(* IEC 61131-3 sources: plc_simulator/services/codesys/POUs (part 2) *)

(* ---- FC_STC_ManualTask.st ---- *)
(* ===========================================================================================
 *  FC_STC_ManualTask — Execute manual transport tasks from gateway
 *
 *  Company : Galvatek part of the John Cockerill Group
 *  Author  : Jarmo Piipponen
 *  Created : 25.03.2026
 *
 * -------------------------------------------------------------------------------------------
 *  For each transporter, checks g_manual_task[vTi].Valid.
 *  If the transporter is idle (Phase=0), validates stations,
 *  calculates transfer time, and inserts a task into the queue
 *  (same pattern as FC_TSK_NoTreatment).
 *  Clears Valid after task is created, or on invalid input.
 *
 *  Called from FB_TSK_Scheduler vPhase 2200 (before NTT).
 *
 * ------------------------------------------------------------------------------------------
 *
 *  Changes:
 *
 *
 *
 *)

FUNCTION FC_STC_ManualTask : BOOL

(* Introduction of Variables ----------------------------------------------------------------*)

VAR_INPUT
  iTimeS                  : LINT;
END_VAR

VAR_IN_OUT
  ioTask                   : ARRAY[1..MAX_TRANSPORTERS] OF UDT_JC_TskQueueType;
END_VAR

VAR_EXTERNAL
  g_manual_task             : ARRAY[1..MAX_TRANSPORTERS] OF UDT_JC_ManualTaskType;
  g_transporter             : ARRAY[1..MAX_TRANSPORTERS] OF UDT_TransporterStatusType;
  g_move                    : ARRAY[1..MAX_TRANSPORTERS] OF UDT_JC_MoveTimesType;
  g_unit                    : ARRAY[1..MAX_UNITS] OF UDT_JC_UnitType;
  Stations                  : ARRAY[MIN_STATION_INDEX..MAX_STATION_INDEX] OF UDT_StationType;
  Transporters              : ARRAY[0..MAX_TRANSPORTERS] OF UDT_TransporterType;
END_VAR

VAR_EXTERNAL CONSTANT
  MAX_TASK_QUEUE            : INT;
  MAX_UNITS                 : INT;
  USED                      : INT;
END_VAR

VAR
  vTi                        : INT;
  vAi                        : INT;
  vSh                        : INT;
  vLift                      : INT;
  vSink                      : INT;
  vCovers                    : BOOL;
  vTransPos                 : INT;
  vTmpMove                  : UDT_JC_MoveTimesType;
  vXferS                    : REAL;
  vTravelToLiftS          : REAL;
  vTaskStart                : LINT;
  vTaskEnd                  : LINT;
END_VAR

FC_STC_ManualTask := TRUE;

FOR vTi := 1 TO MAX_TRANSPORTERS DO
  IF NOT g_manual_task[vTi].Valid THEN
    CONTINUE;
  END_IF;

  vLift := g_manual_task[vTi].LiftStation;
  vSink := g_manual_task[vTi].SinkStation;

  (* Validate station range *)
  IF vLift < MIN_STATION_INDEX OR vLift > MAX_STATION_INDEX
     OR vSink < MIN_STATION_INDEX OR vSink > MAX_STATION_INDEX
     OR vLift = vSink THEN
    g_manual_task[vTi].Valid := FALSE;
    CONTINUE;
  END_IF;

  (* Transporter must be active and idle *)
  (* Transporter must be active and idle or in move-away *)
  IF NOT g_transporter[vTi].IsActive THEN
    CONTINUE;
  END_IF;
  IF g_transporter[vTi].Phase <> 0
     AND NOT (g_transporter[vTi].Phase = 1 AND g_transporter[vTi].Status = 3) THEN
    CONTINUE;  (* keep Valid — retry next cycle *)
  END_IF;

  (* Check vLift station is within transporter TaskArea *)
  vCovers := FALSE;
  FOR vAi := 1 TO 4 DO
    IF Transporters[vTi].TaskArea[vAi].MinLift > 0
       OR Transporters[vTi].TaskArea[vAi].MaxLift > 0 THEN
      IF vLift >= Transporters[vTi].TaskArea[vAi].MinLift
         AND vLift <= Transporters[vTi].TaskArea[vAi].MaxLift THEN
        vCovers := TRUE;
      END_IF;
    END_IF;
  END_FOR;

  IF NOT vCovers THEN
    g_manual_task[vTi].Valid := FALSE;
    CONTINUE;
  END_IF;

  (* Calculate transfer time *)
  vTmpMove := g_move[vTi];
  vXferS := FC_STC_CalcTransferTime(
    iFromStn            := vLift,
    iToStn              := vSink,
    iMove                := vTmpMove,
    iFromDroppingX10   := Stations[vLift].DrippingTime,
    iToDeviceDelayX10 := Stations[vSink].DeviceDelay,
    iDripTrayDelayX10 := Transporters[vTi].DripTrayDelay);

  (* Calculate vTravel-to-vLift: time for transporter to reach vLift station *)
  vTravelToLiftS := 0.0;
  vTransPos := g_transporter[vTi].CurrentStation;
  IF vTransPos > 0 AND vTransPos <> vLift THEN
    vTravelToLiftS := FC_STC_CalcHorizontalTravel(
      iFromStn := vTransPos,
      iToStn   := vLift,
      iMove     := vTmpMove);
  END_IF;

  vTaskStart := iTimeS + REAL_TO_LINT(vTravelToLiftS);
  vTaskEnd   := vTaskStart + REAL_TO_LINT(vXferS);

  (* Check vSink station is free — no unit occupying it *)
  vCovers := TRUE;  (* reuse variable as vSinkFree flag *)
  FOR vSh := 1 TO MAX_UNITS DO
    IF g_unit[vSh].Location = vSink AND g_unit[vSh].Status = USED THEN
      vCovers := FALSE;
    END_IF;
  END_FOR;
  IF NOT vCovers THEN
    g_manual_task[vTi].Valid := FALSE;
    CONTINUE;
  END_IF;

  (* Insert task at queue position 1 *)
  IF ioTask[vTi].Count < MAX_TASK_QUEUE THEN
    FOR vSh := ioTask[vTi].Count TO 1 BY -1 DO
      ioTask[vTi].Queue[vSh + 1] := ioTask[vTi].Queue[vSh];
    END_FOR;
    ioTask[vTi].Queue[1].Unit              := 0;
    ioTask[vTi].Queue[1].Stage             := 0;
    ioTask[vTi].Queue[1].LiftStationTarget := vLift;
    ioTask[vTi].Queue[1].SinkStationTarget := vSink;
    ioTask[vTi].Queue[1].StartTime         := vTaskStart;
    ioTask[vTi].Queue[1].FinishTime        := vTaskEnd;
    ioTask[vTi].Queue[1].CalcTime          := 0;
    ioTask[vTi].Queue[1].MinTime           := 0;
    ioTask[vTi].Queue[1].MaxTime           := 0;
    ioTask[vTi].Queue[1].NttPrimary        := 0;
    ioTask[vTi].Count := ioTask[vTi].Count + 1;
  END_IF;

  g_manual_task[vTi].Valid := FALSE;
END_FOR;

END_FUNCTION

(* ---- FC_STC_NoTreatmentStates.st ---- *)
(* ===========================================================================================
 *  FC_STC_NoTreatmentStates — Non-treatment target state management
 *
 *  Company : Galvatek part of the John Cockerill Group
 *  Author  : Jarmo Piipponen
 *  Created : 25.03.2026
 *
 * -------------------------------------------------------------------------------------------
 *  Manages non-treatment target states for all units.
 *
 *  Structure:
 *  Pass 0 — SNAPSHOT: read unit/batch/station state into vSnap[]
 *  Section 1 — PROCESSED: mark last-stage units as PROCESSED
 *  Section 2 — TO_AVOID: clear occupied next-stage stations
 *  Section 3 — TO_LOADING: route one empty unit to loading
 *
 *  ------------------------------------------------------------------------------------------
 *
 *  Changes:
 *
 *
 *
 *)

FUNCTION FC_STC_NoTreatmentStates : BOOL

(* Introduction of Variables ----------------------------------------------------------------*)

VAR_EXTERNAL CONSTANT
    MAX_UNITS             : INT;
    MAX_STEPS_PER_PROGRAM : INT;
    MAX_STATIONS_PER_STEP : INT;
    MIN_STATION_INDEX     : INT;
    MAX_STATION_INDEX     : INT;
    IN_PROCESS            : INT;
    PROCESSED             : INT;
    NOT_USED              : INT;
    TO_NONE               : INT;
    TO_UNLOAD             : INT;
    TO_AVOID              : INT;
    TO_LOADING            : INT;
    USED                  : INT;
    OP_BUFFER             : INT;
    OP_BUFFER_PROCESSED   : INT;
    OP_LOADING            : INT;
    OP_LOADING_UNLOADING  : INT;
END_VAR

VAR_EXTERNAL
  gUnit              : ARRAY[1..MAX_UNITS] OF UDT_JC_UnitType;
  gBatch             : ARRAY[1..MAX_UNITS] OF UDT_BatchType;
  TreatmentPrograms  : ARRAY[1..MAX_UNITS] OF UDT_TreatmentProgramType;
  Stations           : ARRAY[MIN_STATION_INDEX..MAX_STATION_INDEX] OF UDT_StationType;
  gStationOccupancy  : ARRAY[1..MAX_STATION_INDEX] OF UDT_JC_UnitAtStationType;
  gTimeS             : LINT;
  gProductionQueue   : INT;
  gEventPending      : UDT_JC_EventMsgType;
  gEventPendingValid : BOOL;
END_VAR

VAR
  (* Snapshot *)
  vSnap       : ARRAY[1..MAX_UNITS] OF UDT_JC_UnitSnapType;
  vU          : INT;        (* unit loop index *)
  vHasLoading : BOOL;       (* any unit vAlready has TO_LOADING *)
  (* Section 1+2 *)
  vP          : INT;        (* parallel station loop *)
  vNextStn    : INT;        (* next stage station *)
  vOccUid     : INT;        (* unit_id at an occupied station *)
  vFreeFound  : BOOL;       (* any next-stage station is free *)
  vAvoidUid   : INT;        (* unit to mark TO_AVOID *)
  (* Section 3 *)
  vLoadFree   : BOOL;       (* a loading station is free *)
  vLoadUid    : INT;        (* best candidate for TO_LOADING *)
  vLoadInBuf  : BOOL;       (* current candidate is in buffer *)
  vStk        : INT;        (* station loop *)
  vOp         : INT;        (* station operation code *)
END_VAR

  (* ════════════════════════════════════════════════════════════
     Pass 0 — SNAPSHOT: collect per-unit state in one pass
     ════════════════════════════════════════════════════════════ *)
  vHasLoading := FALSE;

  FOR vU := 1 TO MAX_UNITS DO
    vSnap[vU].IsActive := gUnit[vU].Status <> NOT_USED;
    IF NOT vSnap[vU].IsActive THEN
      CONTINUE;
    END_IF;

    vSnap[vU].Location       := gUnit[vU].Location;
    vSnap[vU].Target       := gUnit[vU].Target;
    vSnap[vU].HasBatch := gBatch[vU].BatchCode <> 0;
    vSnap[vU].BatchState    := gBatch[vU].State;
    vSnap[vU].CurStage := gBatch[vU].CurStage;

    vSnap[vU].OnStation := vSnap[vU].Location >= MIN_STATION_INDEX
                          AND vSnap[vU].Location <= MAX_STATION_INDEX;
    IF vSnap[vU].OnStation THEN
      vSnap[vU].LocationOp    := Stations[vSnap[vU].Location].StationType;
      vSnap[vU].InBuffer := vSnap[vU].LocationOp >= OP_BUFFER AND vSnap[vU].LocationOp <= OP_BUFFER_PROCESSED;
      IF gStationOccupancy[vSnap[vU].Location].ChangeTime > 0 THEN
        vSnap[vU].Elapsed := gTimeS - gStationOccupancy[vSnap[vU].Location].ChangeTime;
      ELSE
        vSnap[vU].Elapsed := 0;
      END_IF;
      IF vSnap[vU].CurStage >= 1 THEN
        vSnap[vU].CalTime := TreatmentPrograms[vU].Steps[vSnap[vU].CurStage].CalTime;
      ELSE
        vSnap[vU].CalTime := 0;
      END_IF;
    ELSE
      vSnap[vU].LocationOp    := 0;
      vSnap[vU].InBuffer := FALSE;
      vSnap[vU].Elapsed   := 0;
      vSnap[vU].CalTime       := 0;
    END_IF;

    IF vSnap[vU].Target = TO_LOADING THEN
      vHasLoading := TRUE;
    END_IF;
  END_FOR;

  (* ════════════════════════════════════════════════════════════
     Section 1 — PROCESSED: mark batch oDone at last treatment stage
     ════════════════════════════════════════════════════════════ *)
  FOR vU := 1 TO MAX_UNITS DO
    IF NOT vSnap[vU].IsActive OR NOT vSnap[vU].HasBatch THEN
      CONTINUE;
    END_IF;
    IF vSnap[vU].BatchState <> IN_PROCESS OR NOT vSnap[vU].OnStation THEN
      CONTINUE;
    END_IF;
    IF vSnap[vU].CurStage >= 1 AND vSnap[vU].CurStage < MAX_STEPS_PER_PROGRAM THEN
      IF vSnap[vU].CurStage >= TreatmentPrograms[vU].StepCount THEN
        IF vSnap[vU].Elapsed > 0 AND vSnap[vU].Elapsed >= DINT_TO_LINT(vSnap[vU].CalTime) THEN
          gBatch[vU].State := PROCESSED;
          vSnap[vU].BatchState   := PROCESSED;  (* update snapshot *)

          (* ── Emit BATCH_COMPLETED event (msg_type=5) ── *)
          IF NOT gEventPendingValid THEN
            gEventPending.MsgType := 5;
            gEventPending.TsHi := LINT_TO_UINT(gTimeS / LINT#65536);
            gEventPending.TsLo := LINT_TO_UINT(gTimeS MOD LINT#65536);
            gEventPending.Payload[1]  := vU;                                  (* unit_id *)
            gEventPending.Payload[2]  := gBatch[vU].BatchCode;               (* batch_code *)
            gEventPending.Payload[3]  := TreatmentPrograms[vU].StepCount;             (* stage_count *)
            gEventPending.Payload[4]  := vSnap[vU].Location;                   (* final_station *)
            gEventPending.Payload[5]  := 0;
            gEventPending.Payload[6]  := 0;
            gEventPending.Payload[7]  := 0;
            gEventPending.Payload[8]  := 0;
            gEventPending.Payload[9]  := 0;
            gEventPending.Payload[10] := 0;
            gEventPending.Payload[11] := 0;
            gEventPending.Payload[12] := 0;
            gEventPendingValid := TRUE;
          END_IF;

          (* Route to unloading station *)
          IF vSnap[vU].Target = TO_NONE THEN
            gUnit[vU].Target := TO_UNLOAD;
            vSnap[vU].Target   := TO_UNLOAD;
          END_IF;
        END_IF;
      END_IF;
    END_IF;
  END_FOR;

  (* ════════════════════════════════════════════════════════════
     Section 2 — TO_AVOID: clear the way to next treatment station
     ════════════════════════════════════════════════════════════ *)
  FOR vU := 1 TO MAX_UNITS DO
    IF NOT vSnap[vU].IsActive OR NOT vSnap[vU].HasBatch THEN
      CONTINUE;
    END_IF;
    IF vSnap[vU].BatchState <> IN_PROCESS THEN
      CONTINUE;
    END_IF;
    IF vSnap[vU].CurStage < 1 OR vSnap[vU].CurStage >= MAX_STEPS_PER_PROGRAM THEN
      CONTINUE;
    END_IF;
    IF vSnap[vU].CurStage >= TreatmentPrograms[vU].StepCount THEN
      CONTINUE;  (* no next stage *)
    END_IF;

    (* — Pass 1: any next-stage station free or being cleared? — *)
    vFreeFound := FALSE;
    vAvoidUid  := 0;
    FOR vP := 0 TO MAX_STATIONS_PER_STEP - 1 DO
      vNextStn := TreatmentPrograms[vU].Steps[vSnap[vU].CurStage + 1].Stations[vP];
      IF vNextStn = 0 THEN
        EXIT;
      END_IF;
      IF vNextStn >= MIN_STATION_INDEX AND vNextStn <= MAX_STATION_INDEX THEN
        IF gStationOccupancy[vNextStn].UnitId = 0 THEN
          vFreeFound := TRUE;
          EXIT;
        END_IF;
        vOccUid := gStationOccupancy[vNextStn].UnitId;
        IF vOccUid >= 1 AND vOccUid <= MAX_UNITS THEN
          IF vSnap[vOccUid].Target = TO_AVOID THEN
            vFreeFound := TRUE;
            EXIT;
          END_IF;
        END_IF;
      END_IF;
    END_FOR;

    (* — Pass 2: all occupied → mark ONE movable unit TO_AVOID — *)
    IF NOT vFreeFound THEN
      FOR vP := 0 TO MAX_STATIONS_PER_STEP - 1 DO
        vNextStn := TreatmentPrograms[vU].Steps[vSnap[vU].CurStage + 1].Stations[vP];
        IF vNextStn = 0 THEN
          EXIT;
        END_IF;
        IF vNextStn >= MIN_STATION_INDEX AND vNextStn <= MAX_STATION_INDEX THEN
          vOccUid := gStationOccupancy[vNextStn].UnitId;
          IF vOccUid >= 1 AND vOccUid <= MAX_UNITS THEN
            IF NOT vSnap[vOccUid].HasBatch AND vSnap[vOccUid].Target = TO_NONE THEN
              vAvoidUid := vOccUid;
              EXIT;
            END_IF;
          END_IF;
        END_IF;
      END_FOR;

      IF vAvoidUid >= 1 THEN
        gUnit[vAvoidUid].Target := TO_AVOID;
        vSnap[vAvoidUid].Target     := TO_AVOID;  (* update snapshot *)
      END_IF;
    END_IF;
  END_FOR;

  (* ════════════════════════════════════════════════════════════
     Section 3 — TO_LOADING: route one empty unit to loading station
     ════════════════════════════════════════════════════════════ *)
  IF gProductionQueue = 1 AND NOT vHasLoading THEN

    (* Check if any loading station is free *)
    vLoadFree := FALSE;
    FOR vStk := MIN_STATION_INDEX TO MAX_STATION_INDEX DO
      vOp := Stations[vStk].StationType;
      IF (vOp = OP_LOADING OR vOp = OP_LOADING_UNLOADING)
         AND gStationOccupancy[vStk].UnitId = 0 THEN
        vLoadFree := TRUE;
        EXIT;
      END_IF;
    END_FOR;

    IF vLoadFree THEN
      vLoadUid    := 0;
      vLoadInBuf := FALSE;
      FOR vU := 1 TO MAX_UNITS DO
        IF vSnap[vU].IsActive AND NOT vSnap[vU].HasBatch
           AND vSnap[vU].Target = TO_NONE AND vSnap[vU].OnStation THEN
          IF vSnap[vU].InBuffer THEN
            IF vLoadUid = 0 THEN
              vLoadUid    := vU;
              vLoadInBuf := TRUE;
            END_IF;
          ELSE
            IF vLoadUid = 0 OR vLoadInBuf THEN
              vLoadUid    := vU;
              vLoadInBuf := FALSE;
            END_IF;
          END_IF;
        END_IF;
      END_FOR;

      IF vLoadUid >= 1 THEN
        gUnit[vLoadUid].Target := TO_LOADING;
      END_IF;
    END_IF; (* vLoadFree *)

  END_IF; (* production_queue AND NOT vHasLoading *)

  FC_STC_NoTreatmentStates := TRUE;

END_FUNCTION

(* ---- FC_STC_ShiftSchedule.st ---- *)
(* ===========================================================================================
 *  FC_STC_ShiftSchedule — Shift schedule + task times
 *
 *  Company : Galvatek part of the John Cockerill Group
 *  Author  : Jarmo Piipponen
 *  Created : 25.03.2026
 *
 * -------------------------------------------------------------------------------------------
 *  Propagates a time shift through one unit's schedule stages
 *  AND through all matching tasks.
 *
 *  Positive iAmount = DELAY (shift later),
 *  Negative iAmount = ADVANCE (shift earlier).
 *
 *  VAR_IN_OUT: ioSchedule, ioTask — caller passes live or
 *  workspace arrays.
 *
 *  ------------------------------------------------------------------------------------------
 *
 *  Changes:
 *
 *
 *
 *)

FUNCTION FC_STC_ShiftSchedule : BOOL

(* Introduction of Variables ----------------------------------------------------------------*)

VAR_INPUT
  iUnit                    : INT;     (* unit index 1..10 *)
  iFromStage              : INT;     (* propagate from this stage onward *)
  iAmount                  : REAL;    (* seconds to shift (+ = later, - = earlier) *)
END_VAR

VAR_IN_OUT  (* array sizes must match GVL_JC_Constants: 10=MAX_UNITS, 3=MAX_TRANSPORTERS *)
  ioSchedule               : ARRAY[1..10] OF UDT_JC_TskScheduleType;
  ioTask                   : ARRAY[1..3] OF UDT_JC_TskQueueType;
END_VAR

VAR_EXTERNAL CONSTANT
    MAX_TRANSPORTERS        : INT;
    MAX_UNITS               : INT;
END_VAR

VAR_EXTERNAL
  g_time_s                  : LINT;
END_VAR

VAR
  sc                        : INT;
  si                        : INT;
  qi                        : INT;
  ti                        : INT;
  vDuration                  : LINT;
END_VAR

FC_STC_ShiftSchedule := TRUE;
IF iUnit < 1 OR iUnit > MAX_UNITS THEN RETURN; END_IF;
IF ABS(iAmount) < 0.001 THEN RETURN; END_IF;

(* -- Shift schedule stages entry/exit times -- *)
sc := ioSchedule[iUnit].StageCount;
FOR si := 1 TO sc DO
  IF si >= 1 AND si <= 30
     AND ioSchedule[iUnit].Stages[si].ProgramStage >= iFromStage THEN
    ioSchedule[iUnit].Stages[si].EntryTime :=
      ioSchedule[iUnit].Stages[si].EntryTime + REAL_TO_LINT(iAmount);
    ioSchedule[iUnit].Stages[si].ExitTime :=
      ioSchedule[iUnit].Stages[si].ExitTime + REAL_TO_LINT(iAmount);
    (* GAP-3: Past-clamp -- don't let EntryTime go before now+1 *)
    IF iAmount < 0.0 AND ioSchedule[iUnit].Stages[si].EntryTime < g_time_s + LINT#1 THEN
      ioSchedule[iUnit].Stages[si].ExitTime := g_time_s + LINT#1
        + (ioSchedule[iUnit].Stages[si].ExitTime - ioSchedule[iUnit].Stages[si].EntryTime);
      ioSchedule[iUnit].Stages[si].EntryTime := g_time_s + LINT#1;
    END_IF;
  END_IF;
END_FOR;

(* -- Shift matching tasks in all transporter queues -- *)
FOR ti := 1 TO MAX_TRANSPORTERS DO
  FOR qi := 1 TO ioTask[ti].Count DO
    IF ioTask[ti].Queue[qi].Unit = iUnit
       AND ioTask[ti].Queue[qi].Stage >= iFromStage THEN
      ioTask[ti].Queue[qi].StartTime :=
        ioTask[ti].Queue[qi].StartTime + REAL_TO_LINT(iAmount);
      ioTask[ti].Queue[qi].FinishTime :=
        ioTask[ti].Queue[qi].FinishTime + REAL_TO_LINT(iAmount);
      (* GAP-3: Past-clamp -- don't let StartTime go before now+1 *)
      IF iAmount < 0.0 AND ioTask[ti].Queue[qi].StartTime < g_time_s + LINT#1 THEN
        vDuration := ioTask[ti].Queue[qi].FinishTime - ioTask[ti].Queue[qi].StartTime;
        ioTask[ti].Queue[qi].StartTime := g_time_s + LINT#1;
        ioTask[ti].Queue[qi].FinishTime := g_time_s + LINT#1 + vDuration;
      END_IF;
    END_IF;
  END_FOR;
END_FOR;

END_FUNCTION

(* ---- FC_STC_SortTasks.st ---- *)
(* ===========================================================================================
 *  FC_STC_SortTasks — Insertion sort task queues by priority
 *
 *  Company : Galvatek part of the John Cockerill Group
 *  Author  : Jarmo Piipponen
 *  Created : 25.03.2026
 *
 * -------------------------------------------------------------------------------------------
 *  Shared FC: both TSK and DEP call this with different arrays.
 *  Priority: emergency (overtime ratio > 1.0) first, then
 *  earliest StartTime.
 *
 *  ------------------------------------------------------------------------------------------
 *
 *  Changes:
 *
 *
 *
 *)

FUNCTION FC_STC_SortTasks : BOOL

(* Introduction of Variables ----------------------------------------------------------------*)

VAR_INPUT
  i_trans                   : INT;    (* 0 = all, 1..3 = specific transporter *)
  i_time_s                  : LINT;
END_VAR

VAR_IN_OUT  (* array sizes must match GVL_JC_Constants: 3=MAX_TRANSPORTERS, 10=MAX_UNITS *)
  io_task                   : ARRAY[1..3] OF UDT_JC_TskQueueType;
  io_batch                  : ARRAY[1..10] OF UDT_BatchType;
END_VAR

VAR_EXTERNAL CONSTANT
    MAX_TRANSPORTERS        : INT;
    MAX_UNITS               : INT;
    IN_PROCESS              : INT;
END_VAR

VAR_EXTERNAL
  g_unit                    : ARRAY[1..MAX_UNITS] OF UDT_JC_UnitType;
END_VAR

VAR
  ti                        : INT;
  t_start                   : INT;
  t_end                     : INT;
  ins_i                     : INT;
  ins_j                     : INT;
  ins_cnt                   : INT;
  tmp_task                  : UDT_JC_TskTaskType;
  tmp_unit                  : INT;
  cur_unit                  : INT;
  tmp_ratio                 : REAL;
  cur_ratio                 : REAL;
  tmp_emerg                 : BOOL;
  cur_emerg                 : BOOL;
  do_shift                  : BOOL;
END_VAR

FC_STC_SortTasks := TRUE;

IF i_trans >= 1 AND i_trans <= 3 THEN
  t_start := i_trans;
  t_end   := i_trans;
ELSE
  t_start := 1;
  t_end   := 3;
END_IF;

FOR ti := t_start TO t_end DO
  ins_cnt := io_task[ti].Count;
  IF ins_cnt >= 2 THEN
    FOR ins_i := 2 TO ins_cnt DO
      tmp_task := io_task[ti].Queue[ins_i];

      tmp_ratio := 0.0;
      tmp_unit  := tmp_task.Unit;
      IF tmp_unit >= 1 AND tmp_unit <= MAX_UNITS THEN
        IF io_batch[tmp_unit].State = IN_PROCESS
           AND tmp_task.Stage >= 1 THEN
          IF io_batch[tmp_unit].CurStage = tmp_task.Stage
             AND g_unit[tmp_unit].location = tmp_task.LiftStationTarget
             AND io_batch[tmp_unit].StartTime > LINT#0
             AND io_batch[tmp_unit].MaxTime > 0 THEN
            tmp_ratio := LINT_TO_REAL(i_time_s - io_batch[tmp_unit].StartTime)
                         / DINT_TO_REAL(io_batch[tmp_unit].MaxTime);
          END_IF;
        END_IF;
      END_IF;
      tmp_emerg := tmp_ratio > 1.0;

      ins_j := 0;
      FOR ins_j := ins_i - 1 TO 1 BY -1 DO
        cur_ratio := 0.0;
        cur_unit  := io_task[ti].Queue[ins_j].Unit;
        IF cur_unit >= 1 AND cur_unit <= MAX_UNITS THEN
          IF io_batch[cur_unit].State = IN_PROCESS
             AND io_task[ti].Queue[ins_j].Stage >= 1 THEN
            IF io_batch[cur_unit].CurStage = io_task[ti].Queue[ins_j].Stage
               AND g_unit[cur_unit].location = io_task[ti].Queue[ins_j].LiftStationTarget
               AND io_batch[cur_unit].StartTime > LINT#0
               AND io_batch[cur_unit].MaxTime > 0 THEN
              cur_ratio := LINT_TO_REAL(i_time_s - io_batch[cur_unit].StartTime)
                           / DINT_TO_REAL(io_batch[cur_unit].MaxTime);
            END_IF;
          END_IF;
        END_IF;
        cur_emerg := cur_ratio > 1.0;

        do_shift := FALSE;
        IF tmp_emerg AND NOT cur_emerg THEN
          do_shift := TRUE;
        ELSIF tmp_emerg AND cur_emerg THEN
          IF tmp_ratio > cur_ratio THEN
            do_shift := TRUE;
          END_IF;
        ELSIF NOT tmp_emerg AND NOT cur_emerg THEN
          IF io_task[ti].Queue[ins_j].StartTime > tmp_task.StartTime THEN
            do_shift := TRUE;
          END_IF;
        END_IF;

        IF NOT do_shift THEN EXIT; END_IF;

        io_task[ti].Queue[ins_j + 1] := io_task[ti].Queue[ins_j];
      END_FOR;

      io_task[ti].Queue[ins_j + 1] := tmp_task;
    END_FOR;
  END_IF;
END_FOR;

END_FUNCTION

(* ---- FC_STC_SwapTasks.st ---- *)
(* ===========================================================================================
 *  FC_STC_SwapTasks — Swap same-station task pairs
 *
 *  Company : Galvatek part of the John Cockerill Group
 *  Author  : Jarmo Piipponen
 *  Created : 25.03.2026
 *
 * -------------------------------------------------------------------------------------------
 *  Shared FC: both TSK and DEP call this with different arrays.
 *  Swaps adjacent tasks on the same transporter when the first
 *  task's sink equals the second task's lift (chain optimization).
 *  Returns swap count.
 *
 *  ------------------------------------------------------------------------------------------
 *
 *  Changes:
 *
 *
 *
 *)

FUNCTION FC_STC_SwapTasks : INT   (* returns swap count *)

(* Introduction of Variables ----------------------------------------------------------------*)

VAR_IN_OUT  (* array sizes must match GVL_JC_Constants: 3=MAX_TRANSPORTERS *)
  ioTask                   : ARRAY[1..3] OF UDT_JC_TskQueueType;
END_VAR

VAR_EXTERNAL CONSTANT
    MAX_TRANSPORTERS        : INT;
END_VAR

VAR
  ti                        : INT;
  qi                        : INT;
  vCnt                       : INT;
  vTmp                       : UDT_JC_TskTaskType;
  vSwaps                     : INT;
END_VAR

vSwaps := 0;

FOR ti := 1 TO MAX_TRANSPORTERS DO
  vCnt := ioTask[ti].Count;
  IF vCnt >= 2 THEN
    FOR qi := 1 TO vCnt - 1 DO
      IF ioTask[ti].Queue[qi].Unit <> ioTask[ti].Queue[qi + 1].Unit
         AND ioTask[ti].Queue[qi].SinkStationTarget = ioTask[ti].Queue[qi + 1].LiftStationTarget THEN
        vTmp := ioTask[ti].Queue[qi];
        ioTask[ti].Queue[qi] := ioTask[ti].Queue[qi + 1];
        ioTask[ti].Queue[qi + 1] := vTmp;
        vSwaps := vSwaps + 1;
      END_IF;
    END_FOR;
  END_IF;
END_FOR;

FC_STC_SwapTasks := vSwaps;

END_FUNCTION

(* ---- FC_STC_TakeOut.st ---- *)
(* FC_STC_TakeOut - Evaluate and trigger idle take-out for transporters
   Uses station-specific TakeOutDelay (seconds) and TakeOutDistance (mm) *)
(* IMPORT_MARKER_2026_04_01_B *)

FUNCTION FC_STC_TakeOut : BOOL

VAR_INPUT
  i_time_s                  : LINT;
END_VAR

VAR
  ti                        : INT;
  current_station           : INT;
  take_out_delay            : INT;
  take_out_dist             : DINT;
  idle_time                 : LINT;
  current_x                 : DINT;
  target_x                  : DINT;
  next_lift_x               : DINT;
  area_center               : DINT;
  dir                       : INT;
  queued_lift_station       : INT;
  time_to_start             : LINT;
  si                        : INT;
  stn_x                     : DINT;
  best_stn                  : INT;
  best_dist                 : DINT;
  dx                        : DINT;
END_VAR

FC_STC_TakeOut := TRUE;

FOR ti := 1 TO MAX_TRANSPORTERS DO

  IF g_transporter[ti].Phase <> 0 THEN CONTINUE; END_IF;
  IF g_transporter[ti].Status <> 3 THEN CONTINUE; END_IF;
  IF NOT g_transporter[ti].IsActive THEN CONTINUE; END_IF;

  current_station := g_transporter[ti].CurrentStation;
  IF current_station < MIN_STATION_INDEX OR current_station > MAX_STATION_INDEX THEN CONTINUE; END_IF;

  take_out_delay := Stations[current_station].TakeOutDelay;
  IF take_out_delay = 0 THEN CONTINUE; END_IF;

  take_out_dist := INT_TO_DINT(Stations[current_station].TakeOutDistance);
  IF take_out_dist <= 0 THEN CONTINUE; END_IF;

  idle_time := i_time_s - g_transporter[ti].IdleStartTime;
  IF idle_time < DINT_TO_LINT(INT_TO_DINT(take_out_delay)) THEN CONTINUE; END_IF;

  (* Defer if next task on SAME station starts soon *)
  IF g_task[ti].Count > 0 THEN
    queued_lift_station := g_task[ti].Queue[1].LiftStationTarget;
    IF queued_lift_station = current_station THEN
      time_to_start := g_task[ti].Queue[1].StartTime - i_time_s;
      IF time_to_start >= 0 AND time_to_start < DINT_TO_LINT(INT_TO_DINT(TAKE_OUT_MIN_WAIT_S)) THEN
        CONTINUE;
      END_IF;
    END_IF;
  END_IF;

  current_x := g_transporter[ti].XPosition;

  (* Determine direction: toward next task or toward area center *)
  IF g_task[ti].Count > 0 THEN
    next_lift_x := Stations[g_task[ti].Queue[1].LiftStationTarget].XPosition;
    IF next_lift_x > current_x THEN
      dir := 1;
    ELSE
      dir := -1;
    END_IF;
  ELSE
    area_center := (Transporters[ti].DrivePosMin + Transporters[ti].DrivePosMax) / 2;
    IF area_center > current_x THEN
      dir := 1;
    ELSE
      dir := -1;
    END_IF;
  END_IF;

  (* Compute minimum target position from TakeOutDistance *)
  target_x := current_x + (INT_TO_DINT(dir) * take_out_dist);

  (* Find nearest station in move direction that is at least take_out_dist away *)
  best_stn := 0;
  best_dist := DINT#2147483647;
  FOR si := MIN_STATION_INDEX TO MIN_STATION_INDEX + CountStations - 1 DO
    stn_x := Stations[si].XPosition;
    IF stn_x = 0 THEN CONTINUE; END_IF;
    (* Station must be in the correct direction and at least take_out_dist from current *)
    IF dir > 0 THEN
      dx := stn_x - current_x;
    ELSE
      dx := current_x - stn_x;
    END_IF;
    IF dx >= take_out_dist AND dx < best_dist THEN
      (* Must be within transporter drive limits *)
      IF stn_x >= Transporters[ti].DrivePosMin AND stn_x <= Transporters[ti].DrivePosMax THEN
        best_dist := dx;
        best_stn := si;
      END_IF;
    END_IF;
  END_FOR;

  IF best_stn > 0 THEN
    target_x := Stations[best_stn].XPosition;
  ELSE
    CONTINUE;  (* no station found in direction — skip take-out *)
  END_IF;

  (* Skip if we can't actually move *)
  IF ABS(target_x - current_x) < 100 THEN CONTINUE; END_IF;

  (* If next task starts soon and take-out would pass over its lift station,
     stop at the lift station instead *)
  IF g_task[ti].Count > 0 THEN
    time_to_start := g_task[ti].Queue[1].StartTime - i_time_s;
    IF time_to_start >= 0 AND time_to_start < DINT_TO_LINT(INT_TO_DINT(TAKE_OUT_MIN_WAIT_S)) THEN
      queued_lift_station := g_task[ti].Queue[1].LiftStationTarget;
      IF queued_lift_station >= MIN_STATION_INDEX AND queued_lift_station <= MAX_STATION_INDEX THEN
        next_lift_x := Stations[queued_lift_station].XPosition;
        (* Check if take-out target is on the other side of lift station *)
        IF dir > 0 AND target_x > next_lift_x AND next_lift_x > current_x THEN
          target_x := next_lift_x;
        ELSIF dir < 0 AND target_x < next_lift_x AND next_lift_x < current_x THEN
          target_x := next_lift_x;
        END_IF;
      END_IF;
    END_IF;
  END_IF;

  (* Re-check: still worth moving? *)
  IF ABS(target_x - current_x) < 100 THEN CONTINUE; END_IF;

  g_transporter[ti].Phase := 1;
  g_transporter[ti].LiftStationTarget := 0;
  g_transporter[ti].SinkStationTarget := 0;
  g_transporter[ti].XDriveTarget := target_x;
  g_transporter[ti].XFinalTarget := target_x;

END_FOR;

FC_STC_TakeOut := TRUE;

END_FUNCTION

(* ---- FC_STC_TrackMoveTimes.st ---- *)
(* ===========================================================================================
 *  FC_STC_TrackMoveTimes — Record vPhase transition timestamps
 *
 *  Company : Galvatek part of the John Cockerill Group
 *  Author  : Jarmo Piipponen
 *  Created : 25.03.2026
 *
 * -------------------------------------------------------------------------------------------
 *  Called from SIM code at each transporter vPhase change.
 *  Uses g_time_100ms (0.1s ticks). On 4→0 completion,
 *  calculates net durations and updates g_move[] with
 *  weighted average: new = (old * 4 + measured) / 5.
 *
 *  ------------------------------------------------------------------------------------------
 *
 *  Changes:
 *
 *
 *
 *)

FUNCTION FC_STC_TrackMoveTimes : BOOL

(* Introduction of Variables ----------------------------------------------------------------*)

VAR_INPUT
  iTrans                   : INT;   (* transporter index 1..MAX_TRANSPORTERS *)
  iPrev                    : INT;   (* previous vPhase *)
  iNew                     : INT;   (* new vPhase *)
END_VAR

VAR_EXTERNAL CONSTANT
    MAX_TRANSPORTERS        : INT;
    MIN_STATION_INDEX        : INT;
    MAX_STATION_INDEX        : INT;
END_VAR

VAR_EXTERNAL
  g_transporter             : ARRAY[1..MAX_TRANSPORTERS] OF UDT_TransporterStatusType;
  Stations                 : ARRAY[MIN_STATION_INDEX..MAX_STATION_INDEX] OF UDT_StationType;
  Transporters                     : ARRAY[0..MAX_TRANSPORTERS] OF UDT_TransporterType;
  g_move                    : ARRAY[1..MAX_TRANSPORTERS] OF UDT_JC_MoveTimesType;
  g_actual_move             : ARRAY[1..MAX_TRANSPORTERS] OF UDT_JC_ActualMoveTimeType;
  g_time_s                  : LINT;
  g_time_100ms              : LINT;
END_VAR

VAR
  t                         : INT;
  vLiftStn                  : INT;
  vSinkStn                  : INT;
  vStartStn                 : INT;
  li                        : INT;   (* lift station index = stn - 100 *)
  si                        : INT;   (* sink station index = stn - 100 *)
  st_i                      : INT;   (* start station index = stn - 100 *)
  raw_lift                  : INT;   (* measured lift vDuration in 0.1s ticks *)
  raw_sink                  : INT;   (* measured sink vDuration in 0.1s ticks *)
  raw_trav1                 : INT;   (* measured vTravel start→lift in 0.1s ticks *)
  raw_trav2                 : INT;   (* measured vTravel lift→sink in 0.1s ticks *)
  drip_x10                  : INT;   (* DrippingTime in 0.1s ticks from lift station *)
  tray_x10                  : INT;   (* DripTrayDelay in 0.1s ticks from transporter config *)
  dev_x10                   : INT;   (* DeviceDelay in 0.1s ticks from sink station *)
END_VAR

t := iTrans;

(* Bounds check *)
IF t < 1 OR t > MAX_TRANSPORTERS THEN
    RETURN;
END_IF;

CASE iPrev OF
    0: (* 0→1 : siirto nostoasemalle alkaa *)
        IF iNew = 1 THEN
            g_actual_move[t].StartStation := g_transporter[t].CurrentStation;
            g_actual_move[t].LiftStation  := g_transporter[t].LiftStationTarget;
            g_actual_move[t].SinkStation  := g_transporter[t].SinkStationTarget;
            g_actual_move[t].ts0 := g_time_100ms;
            g_actual_move[t].Invalidated := FALSE;
        END_IF;
    1: (* 1→2 : nosto alkaa *)
        IF iNew = 2 THEN
            g_actual_move[t].ts1 := g_time_100ms;
        END_IF;
    2: (* 2→3 : siirto laskuasemalle alkaa *)
        IF iNew = 3 THEN
            g_actual_move[t].ts2 := g_time_100ms;
        END_IF;
    3: (* 3→4 : lasku alkaa *)
        IF iNew = 4 THEN
            g_actual_move[t].ts3 := g_time_100ms;
        END_IF;
    4: (* 4→0 : handled after CASE — see below *)
END_CASE;

(* ── Invalidate on anomaly (checked at every vPhase transition) ── *)
IF iNew > 0 THEN
    (* Not in automatic mode: task interrupted *)
    IF g_transporter[t].Status < 4 THEN
        g_actual_move[t].Invalidated := TRUE;
    END_IF;
    (* Transporter fault active *)
    IF g_transporter[t].Fault THEN
        g_actual_move[t].Invalidated := TRUE;
    END_IF;
END_IF;

(* ── 4→0 completion: calculate and update g_move ── *)
IF iPrev = 4 AND iNew = 0 THEN
    g_actual_move[t].ts4 := g_time_100ms;

    (* Only update if all timestamps are valid and transfer was normal *)
    IF g_actual_move[t].ts0 > 0
       AND g_actual_move[t].ts1 > 0
       AND g_actual_move[t].ts2 > 0
       AND g_actual_move[t].ts3 > 0
       AND NOT g_actual_move[t].Invalidated
    THEN
                vLiftStn  := g_actual_move[t].LiftStation;
                vSinkStn  := g_actual_move[t].SinkStation;
                vStartStn := g_actual_move[t].StartStation;
                li   := vLiftStn  - MIN_STATION_INDEX;
                si   := vSinkStn  - MIN_STATION_INDEX;
                st_i := vStartStn - MIN_STATION_INDEX;

                (* Mechanical delays in 0.1s ticks *)
                drip_x10 := Stations[vLiftStn].DrippingTime;
                tray_x10 := Transporters[t].DripTrayDelay;
                dev_x10  := Stations[vSinkStn].DeviceDelay;

                (* Raw durations are vAlready in 0.1s ticks *)
                raw_trav1 := LINT_TO_INT(g_actual_move[t].ts1 - g_actual_move[t].ts0);
                raw_trav2 := LINT_TO_INT(g_actual_move[t].ts3 - g_actual_move[t].ts2);

                (* Net lift = (ts2-ts1) - DrippingTime - DripTrayDelay *)
                raw_lift := LINT_TO_INT(g_actual_move[t].ts2 - g_actual_move[t].ts1)
                            - drip_x10 - tray_x10;

                (* Net sink = (ts4-ts3) - DripTrayDelay - DeviceDelay *)
                raw_sink := LINT_TO_INT(g_actual_move[t].ts4 - g_actual_move[t].ts3)
                            - tray_x10 - dev_x10;

                (* Clamp to minimum 0 *)
  IF raw_lift < 0 THEN raw_lift := 0; END_IF;
  IF raw_sink < 0 THEN raw_sink := 0; END_IF;
  IF raw_trav1 < 0 THEN raw_trav1 := 0; END_IF;
  IF raw_trav2 < 0 THEN raw_trav2 := 0; END_IF;

                (* Bounds check indices *)
                IF li >= 1 AND li <= 30
                   AND si >= 1 AND si <= 30
                   AND st_i >= 1 AND st_i <= 30
                THEN
                    (* Weighted average: new = (old * 4 + measured) / 5 *)

                    (* Lift time at lift station *)
                    g_move[t].LiftTime[li] :=
                        (g_move[t].LiftTime[li] * 4 + raw_lift) / 5;

                    (* Sink time at sink station *)
                    g_move[t].SinkTime[si] :=
                        (g_move[t].SinkTime[si] * 4 + raw_sink) / 5;

                    (* Travel: lift → sink (both directions) — vPhase 3 is always exact station-to-station *)
                    g_move[t].Travel[li].ToTime[si] :=
                        (g_move[t].Travel[li].ToTime[si] * 4 + raw_trav2) / 5;
                    g_move[t].Travel[si].ToTime[li] :=
                        (g_move[t].Travel[si].ToTime[li] * 4 + raw_trav2) / 5;
                END_IF;
            END_IF;
END_IF;

FC_STC_TrackMoveTimes := TRUE;

END_FUNCTION

(* ---- FC_STC_UpdateUnitLocation.st ---- *)
(* ===========================================================================================
 *  FC_STC_UpdateUnitLocation — Update a unit's vLocation
 *
 *  Company : Galvatek part of the John Cockerill Group
 *  Author  : Jarmo Piipponen
 *  Created : 25.03.2026
 *
 * -------------------------------------------------------------------------------------------
 *  Sets g_unit[iUnit].Location to the given new vLocation.
 *  Updates g_station_occupancy[].UnitId + ChangeTime for both old
 *  and new vLocations.
 *
 *  When moving to a station:
 *  - Advances batch CurStage if batch is IN_PROCESS
 *  - Updates batch min/max/cal times from treatment program
 *  - Clears unit target if iNttPrimary = 1
 *
 *  ------------------------------------------------------------------------------------------
 *
 *  Changes:
 *
 *
 *
 *)

FUNCTION FC_STC_UpdateUnitLocation : BOOL

(* Introduction of Variables ----------------------------------------------------------------*)

VAR_INPUT
  iUnit                    : INT;   (* unit number to update *)
  iLocation                : INT;   (* new vLocation: <100 = transporter id, >=100 = station number *)
  iNttPrimary             : INT;   (* 1 = sink is NTT primary → clear target, 0 = don't clear *)
END_VAR

VAR_EXTERNAL CONSTANT
    MAX_UNITS               : INT;
    MAX_TRANSPORTERS        : INT;
    MAX_STEPS_PER_PROGRAM   : INT;
    MIN_STATION_INDEX        : INT;
    MAX_STATION_INDEX        : INT;
    IN_PROCESS              : INT;
    USED                    : INT;
    TO_NONE                 : INT;
END_VAR

VAR_EXTERNAL
  g_unit                    : ARRAY[1..MAX_UNITS] OF UDT_JC_UnitType;
  Stations                 : ARRAY[MIN_STATION_INDEX..MAX_STATION_INDEX] OF UDT_StationType;
  g_station_occupancy             : ARRAY[1..MAX_STATION_INDEX] OF UDT_JC_UnitAtStationType;
  g_batch                   : ARRAY[1..MAX_UNITS] OF UDT_BatchType;
  TreatmentPrograms                 : ARRAY[1..MAX_UNITS] OF UDT_TreatmentProgramType;
  g_transporter             : ARRAY[1..MAX_TRANSPORTERS] OF UDT_TransporterStatusType;
  g_move                    : ARRAY[1..MAX_TRANSPORTERS] OF UDT_JC_MoveTimesType;
  g_time_s                  : LINT;
END_VAR

VAR
  vOldLoc                   : INT;
  vNewStg                   : INT;
END_VAR

IF (iUnit >= 1) AND (iUnit <= MAX_UNITS) THEN
  vOldLoc := g_unit[iUnit].Location;

  (* --- Clear unit_id from old vLocation (unified: transporter or station) --- *)
  IF (vOldLoc >= 1) AND (vOldLoc <= MAX_STATION_INDEX) THEN
    g_station_occupancy[vOldLoc].UnitId     := 0;
    g_station_occupancy[vOldLoc].ChangeTime := g_time_s;
  END_IF;

  (* --- Update unit vLocation --- *)
  g_unit[iUnit].Location := iLocation;

  (* --- Set unit_id on new vLocation (unified: transporter or station) --- *)
  IF (iLocation >= 1) AND (iLocation <= MAX_STATION_INDEX) THEN
    g_station_occupancy[iLocation].UnitId     := iUnit;
    g_station_occupancy[iLocation].ChangeTime := g_time_s;

    (* Station-specific: batch stage advance only when landing on a station *)
    IF (iLocation >= MIN_STATION_INDEX) THEN

    (* Advance batch stage if unit is USED with an active batch *)
    IF (g_unit[iUnit].Status = USED)  (* USED *)
       AND (g_batch[iUnit].BatchCode <> 0)
       AND (g_batch[iUnit].State = IN_PROCESS)
       AND (g_batch[iUnit].CurStage < MAX_STEPS_PER_PROGRAM) THEN
      g_batch[iUnit].CurStage := g_batch[iUnit].CurStage + 1;

      (* Stamp arrival time on new station — used by CalcSchedule for elapsed calculation *)
      g_batch[iUnit].StartTime := g_time_s;

      (* Update batch treatment times from program for the new stage *)
      IF (TreatmentPrograms[iUnit].ProgramId = g_batch[iUnit].ProgId)
         AND (TreatmentPrograms[iUnit].ProgramId > 0) THEN
        vNewStg := g_batch[iUnit].CurStage;
        IF (vNewStg >= 1) AND (vNewStg <= MAX_STEPS_PER_PROGRAM) THEN
          g_batch[iUnit].MinTime := TreatmentPrograms[iUnit].Steps[vNewStg].MinTime;
          g_batch[iUnit].MaxTime := TreatmentPrograms[iUnit].Steps[vNewStg].MaxTime;
          g_batch[iUnit].CalTime := TreatmentPrograms[iUnit].Steps[vNewStg].CalTime;
        END_IF;
      END_IF;
    END_IF;

    (* NOT_PROCESSED batch on station: clear times so UI shows no progress bar *)
    IF (g_batch[iUnit].BatchCode <> 0)
       AND (g_batch[iUnit].State <> IN_PROCESS) THEN
      g_batch[iUnit].MinTime   := 0;
      g_batch[iUnit].CalTime   := 0;
      g_batch[iUnit].MaxTime   := 32000;  (* ~8.9 h cap, INT max safe *)
      g_batch[iUnit].StartTime := g_time_s;
    END_IF;

    (* Clear unit target ONLY when iNttPrimary = 1 (primary NTT destination).
       All other cases: keep target so NTT retries primary later. *)
    IF g_unit[iUnit].Target <> TO_NONE AND iNttPrimary > 0 THEN
      g_unit[iUnit].Target := TO_NONE;  (* primary reached → clear *)
    END_IF;

    END_IF; (* iLocation >= MIN_STATION_INDEX — station-specific block *)
  END_IF; (* iLocation valid *)
END_IF;

FC_STC_UpdateUnitLocation := TRUE;

END_FUNCTION

(* ---- FC_TSK_Analyze.st ---- *)
(* ===========================================================================================
 *  FC_TSK_Analyze — Conflict analysis for task list
 *
 *  Company : Galvatek part of the John Cockerill Group
 *  Author  : Jarmo Piipponen
 *  Created : 25.03.2026
 *
 * -------------------------------------------------------------------------------------------
 *  Read-only analysis: never writes globals.
 *
 *  Three vConflict checks, each stops at first hit:
 *  1. TASK_SEQUENCE
 *  2. CROSS_TRANSPORTER_HANDOFF
 *  3. TRANSPORTER_COLLISION
 *
 *  ------------------------------------------------------------------------------------------
 *
 *  Changes:
 *
 *
 *
 *)

FUNCTION FC_TSK_Analyze : BOOL

(* Introduction of Variables ----------------------------------------------------------------*)

VAR_IN_OUT  (* array sizes must match GVL_JC_Constants: 3=MAX_TRANSPORTERS *)
  ioTask                   : ARRAY[1..3] OF UDT_JC_TskQueueType;
END_VAR

VAR_EXTERNAL CONSTANT
    MAX_TRANSPORTERS        : INT;
    MAX_UNITS               : INT;
    MIN_STATION_INDEX        : INT;
    MAX_STATION_INDEX        : INT;
END_VAR

VAR_EXTERNAL
  Stations                 : ARRAY[MIN_STATION_INDEX..MAX_STATION_INDEX] OF UDT_StationType;
  g_move                    : ARRAY[1..MAX_TRANSPORTERS] OF UDT_JC_MoveTimesType;
END_VAR

VAR_OUTPUT
  oHasConflict            : BOOL;
  oConfType               : INT;     (* 1=TASK_SEQUENCE, 2=COLLISION, 3=HANDOFF *)
  oConfUnit               : INT;
  oConfStage              : INT;
  oConfTrans              : INT;
  oBlockedUnit            : INT;
  oBlockedStage           : INT;
  oDeficit                 : REAL;
  oCheckedCount             : INT;
END_VAR

VAR
  vTi                        : INT;
  vTj                        : INT;
  vQi                        : INT;
  vQj                        : INT;
  vPrevSink                 : INT;
  vNextLift                 : INT;
  vTravelS                  : REAL;
  vGapS                     : REAL;
  vDeficitS                 : REAL;
  vLiftX                    : REAL;
  vSinkX                    : REAL;
  vX1Min                    : REAL;
  vX1Max                    : REAL;
  vX2Min                    : REAL;
  vX2Max                    : REAL;
  vXoStart                  : REAL;
  vXoEnd                    : REAL;
  vToStart                  : LINT;
  vToEnd                    : LINT;
  vLIdx                     : INT;
  vSIdx                     : INT;
  vLiftX2                   : REAL;
  vSinkX2                   : REAL;
  vLIdx2                    : INT;
  vSIdx2                    : INT;
  vCurUnit                  : INT;
  vCurStage                 : INT;
  vFoundNext                : BOOL;
  vRecvPrevEnd             : LINT;
  vRecvPrevSink            : INT;
  vHasRecvPrev             : BOOL;
  vRk                        : INT;
  vRecvPrevUnit            : INT;
  vRecvPrevStg             : INT;
  vRecvTravel               : REAL;
  vRecvEarliest             : LINT;
  vHandoffDeficit           : REAL;
  vTotalTasks               : INT;
  cDeficitTol               : REAL := 1.0;
  vTmpMove                  : UDT_JC_MoveTimesType;
END_VAR

FC_TSK_Analyze := FALSE;
oHasConflict := FALSE;
oConfType    := 0;
oDeficit      := 0.0;
oCheckedCount  := 0;

vTotalTasks := 0;
FOR vTi := 1 TO MAX_TRANSPORTERS DO
  vTotalTasks := vTotalTasks + ioTask[vTi].Count;
END_FOR;
IF vTotalTasks = 0 THEN RETURN; END_IF;

(* CHECK 1: TASK_SEQUENCE *)
FOR vTi := 1 TO MAX_TRANSPORTERS DO
  FOR vQi := 1 TO ioTask[vTi].Count - 1 DO
    IF ioTask[vTi].Queue[vQi].Unit > 0 AND ioTask[vTi].Queue[vQi + 1].Unit > 0 THEN
      vPrevSink := ioTask[vTi].Queue[vQi].SinkStationTarget;
      vNextLift := ioTask[vTi].Queue[vQi + 1].LiftStationTarget;
      vTmpMove := g_move[vTi];
      vTravelS := FC_STC_CalcHorizontalTravel(iFromStn := vPrevSink, iToStn := vNextLift, iMove := vTmpMove);
      vGapS := LINT_TO_REAL(ioTask[vTi].Queue[vQi + 1].StartTime - ioTask[vTi].Queue[vQi].FinishTime);
      vDeficitS := vTravelS - vGapS;
      IF vDeficitS > cDeficitTol THEN
  oHasConflict := TRUE;
  oConfType := 1;
        oConfUnit := ioTask[vTi].Queue[vQi + 1].Unit;
        oConfStage := ioTask[vTi].Queue[vQi + 1].Stage;
        oConfTrans := vTi;
        oBlockedUnit := ioTask[vTi].Queue[vQi].Unit;
        oBlockedStage := ioTask[vTi].Queue[vQi].Stage;
  oDeficit := vDeficitS;
  oCheckedCount := vTotalTasks;
  FC_TSK_Analyze := TRUE; RETURN;
      END_IF;
    END_IF;
  END_FOR;
END_FOR;

(* CHECK 2: CROSS_TRANSPORTER_HANDOFF *)
FOR vTi := 1 TO MAX_TRANSPORTERS DO
  FOR vQi := 1 TO ioTask[vTi].Count DO
    vCurUnit  := ioTask[vTi].Queue[vQi].Unit;
    vCurStage := ioTask[vTi].Queue[vQi].Stage;
    IF vCurUnit > 0 THEN
      vFoundNext := FALSE;
      FOR vTj := 1 TO MAX_TRANSPORTERS DO
        IF vTj <> vTi AND NOT vFoundNext THEN
          FOR vQj := 1 TO ioTask[vTj].Count DO
            IF NOT vFoundNext THEN
              IF ioTask[vTj].Queue[vQj].Unit = vCurUnit
                 AND ioTask[vTj].Queue[vQj].Stage = vCurStage + 1 THEN
                vFoundNext := TRUE;
                vHasRecvPrev := FALSE;
  vRecvPrevEnd := 0;
  vRecvPrevSink := 0;
  vRecvPrevUnit := 0;
  vRecvPrevStg := 0;
                FOR vRk := 1 TO ioTask[vTj].Count DO
                  IF vRk <> vQj THEN
                    IF ioTask[vTj].Queue[vRk].FinishTime <= ioTask[vTj].Queue[vQj].StartTime THEN
                      IF NOT vHasRecvPrev OR ioTask[vTj].Queue[vRk].FinishTime > vRecvPrevEnd THEN
                        vHasRecvPrev := TRUE;
                        vRecvPrevEnd  := ioTask[vTj].Queue[vRk].FinishTime;
                        vRecvPrevSink := ioTask[vTj].Queue[vRk].SinkStationTarget;
                        vRecvPrevUnit := ioTask[vTj].Queue[vRk].Unit;
                        vRecvPrevStg  := ioTask[vTj].Queue[vRk].Stage;
                      END_IF;
                    END_IF;
                  END_IF;
                END_FOR;
                IF vHasRecvPrev THEN
                  vRecvTravel := FC_STC_CalcHorizontalTravel(
                    iFromStn := vRecvPrevSink,
                    iToStn   := ioTask[vTi].Queue[vQi].SinkStationTarget,
                    iMove     := g_move[vTj]);
                  vRecvEarliest := vRecvPrevEnd + REAL_TO_LINT(vRecvTravel);
                  vHandoffDeficit := LINT_TO_REAL(vRecvEarliest - ioTask[vTi].Queue[vQi].FinishTime);
                  IF vHandoffDeficit > cDeficitTol THEN
  oHasConflict := TRUE;
  oConfType := 3;
                    oConfUnit := ioTask[vTi].Queue[vQi].Unit;
                    oConfStage := ioTask[vTi].Queue[vQi].Stage;
                    oConfTrans := vTi;
                    oBlockedUnit := vRecvPrevUnit;
                    oBlockedStage := vRecvPrevStg;
  oDeficit := vHandoffDeficit;
  oCheckedCount := vTotalTasks;
  FC_TSK_Analyze := TRUE; RETURN;
                  END_IF;
                END_IF;
              END_IF;
            END_IF;
          END_FOR;
        END_IF;
      END_FOR;
    END_IF;
  END_FOR;
END_FOR;

(* CHECK 3: TRANSPORTER_COLLISION *)
FOR vTi := 1 TO MAX_TRANSPORTERS DO
  FOR vQi := 1 TO ioTask[vTi].Count DO
    IF ioTask[vTi].Queue[vQi].Unit > 0 THEN
      vLIdx := ioTask[vTi].Queue[vQi].LiftStationTarget - MIN_STATION_INDEX;
      vSIdx := ioTask[vTi].Queue[vQi].SinkStationTarget - MIN_STATION_INDEX;
      IF vLIdx >= 1 AND vLIdx <= 30 THEN
        vLiftX := DINT_TO_REAL(Stations[ioTask[vTi].Queue[vQi].LiftStationTarget].XPosition);
  ELSE vLiftX := 0.0; END_IF;
      IF vSIdx >= 1 AND vSIdx <= 30 THEN
        vSinkX := DINT_TO_REAL(Stations[ioTask[vTi].Queue[vQi].SinkStationTarget].XPosition);
  ELSE vSinkX := 0.0; END_IF;
  IF vLiftX < vSinkX THEN vX1Min := vLiftX;
  vX1Max := vSinkX;
  ELSE vX1Min := vSinkX;
  vX1Max := vLiftX; END_IF;

      FOR vTj := vTi + 1 TO MAX_TRANSPORTERS DO
        FOR vQj := 1 TO ioTask[vTj].Count DO
          IF ioTask[vTj].Queue[vQj].Unit > 0 THEN
            vLIdx2 := ioTask[vTj].Queue[vQj].LiftStationTarget - MIN_STATION_INDEX;
            vSIdx2 := ioTask[vTj].Queue[vQj].SinkStationTarget - MIN_STATION_INDEX;
            IF vLIdx2 >= 1 AND vLIdx2 <= 30 THEN
              vLiftX2 := DINT_TO_REAL(Stations[ioTask[vTj].Queue[vQj].LiftStationTarget].XPosition);
  ELSE vLiftX2 := 0.0; END_IF;
            IF vSIdx2 >= 1 AND vSIdx2 <= 30 THEN
              vSinkX2 := DINT_TO_REAL(Stations[ioTask[vTj].Queue[vQj].SinkStationTarget].XPosition);
  ELSE vSinkX2 := 0.0; END_IF;
  IF vLiftX2 < vSinkX2 THEN vX2Min := vLiftX2;
  vX2Max := vSinkX2;
  ELSE vX2Min := vSinkX2;
  vX2Max := vLiftX2; END_IF;

  vXoStart := vX1Min; IF vX2Min > vXoStart THEN vXoStart := vX2Min; END_IF;
  vXoEnd := vX1Max; IF vX2Max < vXoEnd THEN vXoEnd := vX2Max; END_IF;

            IF vXoStart < vXoEnd THEN
              vToStart := ioTask[vTi].Queue[vQi].StartTime;
  IF ioTask[vTj].Queue[vQj].StartTime > vToStart THEN vToStart := ioTask[vTj].Queue[vQj].StartTime; END_IF;
              vToEnd := ioTask[vTi].Queue[vQi].FinishTime;
  IF ioTask[vTj].Queue[vQj].FinishTime < vToEnd THEN vToEnd := ioTask[vTj].Queue[vQj].FinishTime; END_IF;

              IF vToStart < vToEnd THEN
                vDeficitS := LINT_TO_REAL(vToEnd - vToStart) + 2.0;
  oHasConflict := TRUE;
  oConfType := 2;
                IF ioTask[vTi].Queue[vQi].StartTime <= ioTask[vTj].Queue[vQj].StartTime THEN
                  oConfUnit := ioTask[vTj].Queue[vQj].Unit;
                  oConfStage := ioTask[vTj].Queue[vQj].Stage;
                  oConfTrans := vTj;
                  oBlockedUnit := ioTask[vTi].Queue[vQi].Unit;
                  oBlockedStage := ioTask[vTi].Queue[vQi].Stage;
                ELSE
                  oConfUnit := ioTask[vTi].Queue[vQi].Unit;
                  oConfStage := ioTask[vTi].Queue[vQi].Stage;
                  oConfTrans := vTi;
                  oBlockedUnit := ioTask[vTj].Queue[vQj].Unit;
                  oBlockedStage := ioTask[vTj].Queue[vQj].Stage;
                END_IF;
  oDeficit := vDeficitS;
  oCheckedCount := vTotalTasks;
  FC_TSK_Analyze := TRUE; RETURN;
              END_IF;
            END_IF;
          END_IF;
        END_FOR;
      END_FOR;
    END_IF;
  END_FOR;
END_FOR;

oCheckedCount := vTotalTasks;

END_FUNCTION

(* ---- FC_TSK_NoTreatment.st ---- *)
(* ===========================================================================================
 *  FC_TSK_NoTreatment — Create no-treatment transfer tasks
 *
 *  Company : Galvatek part of the John Cockerill Group
 *  Author  : Jarmo Piipponen
 *  Created : 25.03.2026
 *
 * -------------------------------------------------------------------------------------------
 *  Scans units with a target and creates transfer tasks
 *  using the g_ntt destination table.
 *
 *  VAR_IN_OUT: ioTask — only mutable array (inserts NTT tasks).
 *  All other globals are read-only via VAR_EXTERNAL.
 *
 *  ------------------------------------------------------------------------------------------
 *
 *  Changes:
 *
 *
 *
 *)

FUNCTION FC_TSK_NoTreatment : BOOL

(* Introduction of Variables ----------------------------------------------------------------*)

VAR_INPUT
  iTimeS                  : LINT;
END_VAR

VAR_IN_OUT  (* array sizes must match GVL_JC_Constants: 3=MAX_TRANSPORTERS *)
  ioTask                   : ARRAY[1..3] OF UDT_JC_TskQueueType;
END_VAR

VAR_EXTERNAL CONSTANT
    MAX_TRANSPORTERS        : INT;
    MAX_STATIONS_PER_STEP   : INT;
    MIN_STATION_INDEX        : INT;
    MAX_STATION_INDEX        : INT;
    MAX_UNITS               : INT;
    MAX_TASK_QUEUE          : INT;
    SCH_DISPATCH_MARGIN_S   : REAL;
    NOT_PROCESSED           : INT;
    PROCESSED               : INT;
    USED                    : INT;
END_VAR

VAR_EXTERNAL
  g_unit                    : ARRAY[1..MAX_UNITS] OF UDT_JC_UnitType;
  g_batch                   : ARRAY[1..MAX_UNITS] OF UDT_BatchType;
  g_ntt                     : ARRAY[1..MAX_TRANSPORTERS] OF UDT_JC_NttTransporterType;
  g_transporter             : ARRAY[1..MAX_TRANSPORTERS] OF UDT_TransporterStatusType;
  Stations                 : ARRAY[MIN_STATION_INDEX..MAX_STATION_INDEX] OF UDT_StationType;
  g_station_occupancy             : ARRAY[1..MAX_STATION_INDEX] OF UDT_JC_UnitAtStationType;
  Transporters                     : ARRAY[0..MAX_TRANSPORTERS] OF UDT_TransporterType;
  g_move                    : ARRAY[1..MAX_TRANSPORTERS] OF UDT_JC_MoveTimesType;
END_VAR

VAR
  ui                        : INT;
  vLoc                       : INT;
  tgt                       : INT;
  cov_t                     : INT;
  ai                        : INT;
  vCovers                    : BOOL;
  oDone                      : BOOL;
  vDest                      : UDT_JC_NttDestType;
  vNttIdx                   : INT;
  vOnPrimary                : BOOL;
  vOnFallback               : BOOL;
  vPrimaryFree              : BOOL;
  vDestStn                  : INT;
  si                        : INT;
  vStationIdx               : INT;
  vStnFree                  : BOOL;
  uj                        : INT;
  ti                        : INT;
  vAlready                   : BOOL;
  qi2                       : INT;
  vXferS                    : REAL;
  vTaskStart                : LINT;
  vTaskEnd                  : LINT;
  vSlotStart                : LINT;
  vTmpMove                  : UDT_JC_MoveTimesType;
  vSlotEnd                  : LINT;
  latest_end                : LINT;
  vTravelFromSink          : REAL;
  vTravelToLiftS          : REAL;
  vTransPos                 : INT;
  vNttDuration              : LINT;
  vSlotOk                   : BOOL;
  sh                        : INT;

  (* Idle-stretch: extend blocking batch CalTime to make room for NTT -----------------------*)
  vStretchPending           : BOOL;
  vStretchUnitId           : INT;
  vStretchDeficit           : DINT;
  vStretchAvail             : DINT;

  (* Multi-transporter shared-vArea idle check -----------------------------------------------*)
  ot                        : INT;
  oq                        : INT;
  vOverlapConflict          : BOOL;
  vDestX                    : DINT;
  vAvoidDist                : DINT;
  cov_min_x                 : DINT;
  cov_max_x                 : DINT;
  ot_min_x                  : DINT;
  ot_max_x                  : DINT;
  zone_min_x                : DINT;
  zone_max_x                : DINT;
  danger_min                : DINT;
  danger_max                : DINT;
  (* Shared-vArea timing: NTT split into own-vArea + shared-vArea portions ---------------------*)
  vLocIdx                   : INT;
  vLocX                     : DINT;
  phase2_s                  : REAL;
  vSharedEntry              : LINT;
  vSharedTime               : REAL;
  ot_idle_ok                : BOOL;
  ot_idle_start             : LINT;
  ot_idle_end               : LINT;
  ot_next_lift              : INT;
  ot_dispatch_from          : INT;
  ot_travel_to_next         : REAL;

  (* Idle-stretch for other transporter: widen idle gap by extending blocker CalTime --------*)
  ot_stretch_pending        : BOOL;
  ot_stretch_unit_id        : INT;
  ot_stretch_deficit        : DINT;
  ot_stretch_avail          : DINT;
  ot_stretch_need           : LINT;
  ot_stretch_ok             : BOOL;
END_VAR

FC_TSK_NoTreatment := TRUE;

FOR ui := 1 TO MAX_UNITS DO
  tgt := g_unit[ui].Target;
  vLoc := g_unit[ui].Location;

  IF tgt >= 1 AND tgt <= 5 AND vLoc >= MIN_STATION_INDEX THEN

    IF tgt = 3 AND (g_batch[ui].BatchCode = 0 OR g_batch[ui].State <> NOT_PROCESSED) THEN
      CONTINUE;
    END_IF;

    vAlready := FALSE;
    FOR ti := 1 TO MAX_TRANSPORTERS DO
      IF NOT vAlready THEN
        IF g_transporter[ti].Phase > 0 AND g_station_occupancy[ti].UnitId = ui THEN
          vAlready := TRUE;
        END_IF;
        FOR qi2 := 1 TO ioTask[ti].Count DO
          IF NOT vAlready THEN
            IF ioTask[ti].Queue[qi2].Unit = ui THEN
              vAlready := TRUE;
            END_IF;
          END_IF;
        END_FOR;
      END_IF;
    END_FOR;

    IF NOT vAlready THEN

    oDone := FALSE;
    FOR cov_t := 1 TO MAX_TRANSPORTERS DO
      IF NOT oDone THEN

      vCovers := FALSE;
      FOR ai := 1 TO 4 DO
        IF NOT vCovers THEN
          IF Transporters[cov_t].TaskArea[ai].MinLift > 0 OR Transporters[cov_t].TaskArea[ai].MaxLift > 0 THEN
            IF vLoc >= Transporters[cov_t].TaskArea[ai].MinLift AND vLoc <= Transporters[cov_t].TaskArea[ai].MaxLift THEN
              vCovers := TRUE;
            END_IF;
          END_IF;
        END_IF;
      END_FOR;

      IF vCovers AND g_transporter[cov_t].IsActive
         AND (g_transporter[cov_t].Phase = 0 OR tgt = 5) THEN

        IF tgt = 2 THEN
          IF g_batch[ui].BatchCode = 0 THEN vNttIdx := 6;
          ELSIF g_batch[ui].State = PROCESSED THEN vNttIdx := 8;
  ELSE vNttIdx := 7; END_IF;
        ELSIF tgt = 3 THEN vNttIdx := 7;
  ELSE vNttIdx := tgt; END_IF;

        vDest := g_ntt[cov_t].Target[vNttIdx];

        vOnPrimary := FALSE;
        FOR si := 1 TO vDest.StationCount DO
  IF vDest.Stations[si] = vLoc THEN vOnPrimary := TRUE; END_IF;
        END_FOR;

        IF NOT vOnPrimary THEN

          vOnFallback := FALSE;
          FOR si := 1 TO vDest.FallbackCount DO
  IF vDest.FallbackStations[si] = vLoc THEN vOnFallback := TRUE; END_IF;
          END_FOR;

          vPrimaryFree := FALSE;
          FOR si := 1 TO vDest.StationCount DO
            vStationIdx := vDest.Stations[si];
            IF vStationIdx <> vLoc AND vStationIdx >= MIN_STATION_INDEX AND vStationIdx <= MAX_STATION_INDEX THEN
              vStnFree := TRUE;
              FOR uj := 1 TO MAX_UNITS DO
  IF g_unit[uj].Location = vStationIdx AND g_unit[uj].Status = USED THEN vStnFree := FALSE; END_IF;
              END_FOR;
  IF vStnFree THEN vPrimaryFree := TRUE; END_IF;
            END_IF;
          END_FOR;

          vDestStn := 0;

          IF vOnFallback AND NOT vPrimaryFree THEN
            vDestStn := 0;
          ELSIF vOnFallback AND vPrimaryFree THEN
            FOR si := 1 TO vDest.StationCount DO
              IF vDestStn = 0 THEN
                vStationIdx := vDest.Stations[si];
                IF vStationIdx <> vLoc AND vStationIdx >= MIN_STATION_INDEX AND vStationIdx <= MAX_STATION_INDEX THEN
                  vStnFree := TRUE;
                  FOR uj := 1 TO MAX_UNITS DO
  IF g_unit[uj].Location = vStationIdx AND g_unit[uj].Status = USED THEN vStnFree := FALSE; END_IF;
                  END_FOR;
  IF vStnFree THEN vDestStn := vStationIdx; END_IF;
                END_IF;
              END_IF;
            END_FOR;
          ELSE
            FOR si := 1 TO vDest.StationCount DO
              IF vDestStn = 0 THEN
                vStationIdx := vDest.Stations[si];
                IF vStationIdx <> vLoc AND vStationIdx >= MIN_STATION_INDEX AND vStationIdx <= MAX_STATION_INDEX THEN
                  vStnFree := TRUE;
                  FOR uj := 1 TO MAX_UNITS DO
  IF g_unit[uj].Location = vStationIdx AND g_unit[uj].Status = USED THEN vStnFree := FALSE; END_IF;
                  END_FOR;
  IF vStnFree THEN vDestStn := vStationIdx; END_IF;
                END_IF;
              END_IF;
            END_FOR;

            IF vDestStn = 0 THEN
              FOR si := 1 TO vDest.FallbackCount DO
                IF vDestStn = 0 THEN
                  vStationIdx := vDest.FallbackStations[si];
                  IF vStationIdx <> vLoc AND vStationIdx >= MIN_STATION_INDEX AND vStationIdx <= MAX_STATION_INDEX THEN
                    vStnFree := TRUE;
                    FOR uj := 1 TO MAX_UNITS DO
  IF g_unit[uj].Location = vStationIdx AND g_unit[uj].Status = USED THEN vStnFree := FALSE; END_IF;
                    END_FOR;
  IF vStnFree THEN vDestStn := vStationIdx; END_IF;
                  END_IF;
                END_IF;
              END_FOR;
            END_IF;
          END_IF;

          IF vDestStn > 0 THEN
            vTmpMove := g_move[cov_t];
            vXferS := FC_STC_CalcTransferTime(
              iFromStn            := vLoc,
              iToStn              := vDestStn,
              iMove                := vTmpMove,
              i_from_dropping_x10   := Stations[vLoc].DrippingTime,
              i_to_device_delay_x10 := Stations[vDestStn].DeviceDelay,
              iDripTrayDelayX10 := Transporters[cov_t].DripTrayDelay);

            (* ── Travel-to: time for transporter to reach lift station ── *)
            vTravelToLiftS := 0.0;
            IF g_transporter[cov_t].Phase = 0 THEN
              vTransPos := g_transporter[cov_t].CurrentStation;
            ELSE
              vTransPos := g_transporter[cov_t].SinkStationTarget;
            END_IF;
            IF vTransPos > 0 AND vTransPos <> vLoc THEN
              vTravelToLiftS := FC_STC_CalcHorizontalTravel(
                iFromStn := vTransPos,
                iToStn   := vLoc,
                iMove     := vTmpMove);
            END_IF;

            vTaskStart := iTimeS + REAL_TO_LINT(vTravelToLiftS);
            vTaskEnd   := vTaskStart + REAL_TO_LINT(vXferS);
            vNttDuration := vTaskEnd - vTaskStart;

            vSlotOk := FALSE;
            vStretchPending := FALSE;
            ot_stretch_pending := FALSE;

            IF ioTask[cov_t].Count = 0 THEN
              vSlotOk := TRUE;
            ELSE
              IF ioTask[cov_t].Queue[1].StartTime > vTaskStart THEN
                vSlotStart := vTaskStart;
                vSlotEnd   := ioTask[cov_t].Queue[1].StartTime;
                vTravelFromSink := FC_STC_CalcHorizontalTravel(
                  iFromStn := vDestStn,
                  iToStn   := ioTask[cov_t].Queue[1].LiftStationTarget,
                  iMove     := g_move[cov_t]);
                latest_end := vSlotEnd - REAL_TO_LINT(vTravelFromSink) - 1;
                IF vTaskStart >= vSlotStart AND vTaskEnd <= latest_end THEN
                  vSlotOk := TRUE;
                END_IF;

                (* ── Idle-stretch: NTT slightly too long for idle window ──
                   Check if the blocking batch's treatment CalTime can be
                   extended (up to MaxTime) to widen the idle gap.  Only flag
                   the intent here; the actual g_batch write happens after
                   the multi-transporter overlap check passes. *)
                IF NOT vSlotOk AND latest_end > 0 THEN
                  vStretchDeficit := LINT_TO_DINT(vTaskEnd - latest_end);
                  IF vStretchDeficit > 0 THEN
                    vStretchUnitId := ioTask[cov_t].Queue[1].Unit;
                    IF vStretchUnitId >= 1 AND vStretchUnitId <= MAX_UNITS THEN
                      vStretchAvail := g_batch[vStretchUnitId].MaxTime
                                     - g_batch[vStretchUnitId].CalTime;
                      IF vStretchAvail >= vStretchDeficit THEN
                        vStretchPending := TRUE;
                        vSlotOk := TRUE;
                      END_IF;
                    END_IF;
                  END_IF;
                END_IF;
              END_IF;
            END_IF;

            IF NOT vSlotOk THEN
              IF ioTask[cov_t].Count > 0
                 AND ioTask[cov_t].Queue[1].SinkStationTarget = vLoc THEN
                vSlotOk := TRUE;
              ELSE
                vDestStn := 0;
              END_IF;
            END_IF;
          END_IF;

          (* ── Multi-transporter shared-vArea idle check ──
             If vDestStn is on the shared drive vArea between two transporters,
             the other transporter must have an idle window covering the time
             when THIS transporter is physically on the shared vArea.

             NTT transfer phases:
               Phase 2: lift + drip + tray  (nostin on vielä lift-asemalla)
               Phase 3: horizontal vTravel   (nostin liikkuu kohti vDest)
               Phase 4: lower + tray + dev  (nostin on vDest-asemalla)

             If lift station is NOT on shared vArea:
               vSharedEntry = vTaskStart + phase2_s  (vTravel starts)
               vSharedTime  = vXferS - phase2_s
             If lift station IS on shared vArea:
               vSharedEntry = vTaskStart  (vAlready there)
               vSharedTime  = vXferS
          *)
          IF vDestStn > 0 THEN
            vOverlapConflict := FALSE;
            vDestX := Stations[vDestStn].XPosition;
            vAvoidDist := Transporters[cov_t].AvoidanceWidth;
            cov_min_x := Transporters[cov_t].DrivePosMin;
            cov_max_x := Transporters[cov_t].DrivePosMax;

            FOR ot := 1 TO MAX_TRANSPORTERS DO
              IF ot <> cov_t AND NOT vOverlapConflict
                 AND g_transporter[ot].IsActive THEN
                ot_min_x := Transporters[ot].DrivePosMin;
                ot_max_x := Transporters[ot].DrivePosMax;

                IF cov_min_x > ot_min_x THEN zone_min_x := cov_min_x;
  ELSE zone_min_x := ot_min_x; END_IF;
                IF cov_max_x < ot_max_x THEN zone_max_x := cov_max_x;
  ELSE zone_max_x := ot_max_x; END_IF;

                IF zone_min_x >= zone_max_x THEN CONTINUE; END_IF;
                IF vDestX < zone_min_x OR vDestX > zone_max_x THEN CONTINUE; END_IF;

                danger_min := zone_min_x - vAvoidDist;
                danger_max := zone_max_x + vAvoidDist;

                (* ── Calculate shared-vArea entry time and vDuration ── *)
                vLocX := Stations[vLoc].XPosition;
                IF vLocX >= danger_min AND vLocX <= danger_max THEN
                  vSharedEntry := vTaskStart;
                  vSharedTime  := vXferS;
                ELSE
                  vLocIdx := vLoc - MIN_STATION_INDEX;
                  IF vLocIdx >= 1 AND vLocIdx <= 25 THEN
                    phase2_s := INT_TO_REAL(g_move[cov_t].LiftTime[vLocIdx]) / 10.0
                              + INT_TO_REAL(Stations[vLoc].DrippingTime) / 10.0
                              + INT_TO_REAL(Transporters[cov_t].DripTrayDelay) / 10.0;
                  ELSE
                    phase2_s := 0.0;
                  END_IF;
                  vSharedEntry := vTaskStart + REAL_TO_LINT(phase2_s);
                  vSharedTime  := vXferS - phase2_s;
  IF vSharedTime < 1.0 THEN vSharedTime := 1.0; END_IF;
                END_IF;

                (* ── Check: does other transporter have an idle window
                     that starts ≤ vSharedEntry and lasts ≥ vSharedTime? ── *)
                ot_idle_ok := FALSE;

                IF ioTask[ot].Count = 0 AND g_transporter[ot].Phase = 0 THEN
                  ot_idle_ok := TRUE;
                ELSIF ioTask[ot].Count = 0
                      AND g_transporter[ot].Phase >= 1
                      AND g_transporter[ot].Phase <= 4 THEN
                  (* Transporter executing task, nothing queued after.
                     Idle starts at current task finish. *)
                  ot_idle_start := g_transporter[ot].CurrentTaskFinishTime;
                  IF ot_idle_start <= vSharedEntry THEN
                    ot_idle_ok := TRUE;
                  END_IF;
                ELSE
                  IF ioTask[ot].Count > 0 THEN
                    IF g_transporter[ot].Phase >= 1 AND g_transporter[ot].Phase <= 4 THEN
                      (* Idle gap: current task finish → next queued start *)
                      ot_idle_start := g_transporter[ot].CurrentTaskFinishTime;
                      ot_dispatch_from := g_transporter[ot].SinkStationTarget;
                    ELSE
                      ot_idle_start := vTaskStart;
                      ot_dispatch_from := g_transporter[ot].CurrentStation;
                    END_IF;
                    ot_next_lift := ioTask[ot].Queue[1].LiftStationTarget;
                    ot_travel_to_next := 0.0;
                    IF ot_dispatch_from > 0
                       AND ot_next_lift > 0
                       AND ot_dispatch_from <> ot_next_lift THEN
                      ot_travel_to_next := FC_STC_CalcHorizontalTravel(
                        iFromStn := ot_dispatch_from,
                        iToStn   := ot_next_lift,
                        iMove     := g_move[ot]);
                    END_IF;
                    ot_idle_end := ioTask[ot].Queue[1].StartTime
                                 - REAL_TO_LINT(ot_travel_to_next)
                                 - REAL_TO_LINT(SCH_DISPATCH_MARGIN_S);
                    IF ot_idle_end < ot_idle_start THEN
                      ot_idle_end := ot_idle_start;
                    END_IF;
                    IF ot_idle_start <= vSharedEntry
                       AND ot_idle_end >= vSharedEntry + REAL_TO_LINT(vSharedTime) THEN
                      ot_idle_ok := TRUE;
                    END_IF;
                  END_IF;

                  IF NOT ot_idle_ok THEN
                    FOR oq := 1 TO ioTask[ot].Count - 1 DO
                      IF NOT ot_idle_ok THEN
                        ot_idle_start := ioTask[ot].Queue[oq].FinishTime;
                        ot_dispatch_from := ioTask[ot].Queue[oq].SinkStationTarget;
                        ot_next_lift := ioTask[ot].Queue[oq + 1].LiftStationTarget;
                        ot_travel_to_next := 0.0;
                        IF ot_dispatch_from > 0
                           AND ot_next_lift > 0
                           AND ot_dispatch_from <> ot_next_lift THEN
                          ot_travel_to_next := FC_STC_CalcHorizontalTravel(
                            iFromStn := ot_dispatch_from,
                            iToStn   := ot_next_lift,
                            iMove     := g_move[ot]);
                        END_IF;
                        ot_idle_end := ioTask[ot].Queue[oq + 1].StartTime
                                     - REAL_TO_LINT(ot_travel_to_next)
                                     - REAL_TO_LINT(SCH_DISPATCH_MARGIN_S);
                        IF ot_idle_end < ot_idle_start THEN
                          ot_idle_end := ot_idle_start;
                        END_IF;
                        IF ot_idle_start <= vSharedEntry
                           AND ot_idle_end >= vSharedEntry + REAL_TO_LINT(vSharedTime) THEN
                          ot_idle_ok := TRUE;
                        END_IF;
                      END_IF;
                    END_FOR;
                  END_IF;

                  IF NOT ot_idle_ok AND ioTask[ot].Count > 0 THEN
                    ot_idle_start := ioTask[ot].Queue[ioTask[ot].Count].FinishTime;
                    IF ot_idle_start <= vSharedEntry THEN
                      ot_idle_ok := TRUE;
                    END_IF;
                  END_IF;
                END_IF;

                IF NOT ot_idle_ok THEN
                  (* ── Idle-stretch for other transporter ──
                     Try to widen the nearest idle gap by extending the
                     blocking batch CalTime (up to MaxTime).  Only tasks
                     with Stage > 0 (regular, not NTT) are candidates. *)
                  ot_stretch_ok := FALSE;

                  (* Try gap before first task *)
                  IF ioTask[ot].Count > 0
                     AND ioTask[ot].Queue[1].Stage > 0 THEN
                    IF g_transporter[ot].Phase >= 1 AND g_transporter[ot].Phase <= 4 THEN
                      ot_idle_start := g_transporter[ot].CurrentTaskFinishTime;
                      ot_dispatch_from := g_transporter[ot].SinkStationTarget;
                    ELSE
                      ot_idle_start := vTaskStart;
                      ot_dispatch_from := g_transporter[ot].CurrentStation;
                    END_IF;
                    ot_next_lift := ioTask[ot].Queue[1].LiftStationTarget;
                    ot_travel_to_next := 0.0;
                    IF ot_dispatch_from > 0
                       AND ot_next_lift > 0
                       AND ot_dispatch_from <> ot_next_lift THEN
                      ot_travel_to_next := FC_STC_CalcHorizontalTravel(
                        iFromStn := ot_dispatch_from,
                        iToStn   := ot_next_lift,
                        iMove     := g_move[ot]);
                    END_IF;
                    ot_idle_end := ioTask[ot].Queue[1].StartTime
                                 - REAL_TO_LINT(ot_travel_to_next)
                                 - REAL_TO_LINT(SCH_DISPATCH_MARGIN_S);
                    IF ot_idle_end < ot_idle_start THEN
                      ot_idle_end := ot_idle_start;
                    END_IF;

                    IF ot_idle_start <= vSharedEntry
                       AND ot_idle_end > vSharedEntry THEN
                      ot_stretch_need := vSharedEntry
                                       + REAL_TO_LINT(vSharedTime)
                                       - ot_idle_end;
                      IF ot_stretch_need > LINT#0 THEN
                        ot_stretch_unit_id := ioTask[ot].Queue[1].Unit;
                        IF ot_stretch_unit_id >= 1
                           AND ot_stretch_unit_id <= MAX_UNITS THEN
                          ot_stretch_avail :=
                            g_batch[ot_stretch_unit_id].MaxTime
                          - g_batch[ot_stretch_unit_id].CalTime;
                          IF ot_stretch_avail >= LINT_TO_DINT(ot_stretch_need) THEN
                            ot_stretch_deficit := LINT_TO_DINT(ot_stretch_need);
                            ot_stretch_pending := TRUE;
                            ot_stretch_ok      := TRUE;
                          END_IF;
                        END_IF;
                      END_IF;
                    END_IF;
                  END_IF;

                  (* Try gaps between tasks *)
                  IF NOT ot_stretch_ok THEN
                    FOR oq := 1 TO ioTask[ot].Count - 1 DO
                      IF NOT ot_stretch_ok
                         AND ioTask[ot].Queue[oq + 1].Stage > 0 THEN
                        ot_idle_start := ioTask[ot].Queue[oq].FinishTime;
                        ot_dispatch_from := ioTask[ot].Queue[oq].SinkStationTarget;
                        ot_next_lift := ioTask[ot].Queue[oq + 1].LiftStationTarget;
                        ot_travel_to_next := 0.0;
                        IF ot_dispatch_from > 0
                           AND ot_next_lift > 0
                           AND ot_dispatch_from <> ot_next_lift THEN
                          ot_travel_to_next := FC_STC_CalcHorizontalTravel(
                            iFromStn := ot_dispatch_from,
                            iToStn   := ot_next_lift,
                            iMove     := g_move[ot]);
                        END_IF;
                        ot_idle_end := ioTask[ot].Queue[oq + 1].StartTime
                                     - REAL_TO_LINT(ot_travel_to_next)
                                     - REAL_TO_LINT(SCH_DISPATCH_MARGIN_S);
                        IF ot_idle_end < ot_idle_start THEN
                          ot_idle_end := ot_idle_start;
                        END_IF;

                        IF ot_idle_start <= vSharedEntry
                           AND ot_idle_end > vSharedEntry THEN
                          ot_stretch_need := vSharedEntry
                                           + REAL_TO_LINT(vSharedTime)
                                           - ot_idle_end;
                          IF ot_stretch_need > LINT#0 THEN
                            ot_stretch_unit_id := ioTask[ot].Queue[oq + 1].Unit;
                            IF ot_stretch_unit_id >= 1
                               AND ot_stretch_unit_id <= MAX_UNITS THEN
                              ot_stretch_avail :=
                                g_batch[ot_stretch_unit_id].MaxTime
                              - g_batch[ot_stretch_unit_id].CalTime;
                              IF ot_stretch_avail >= LINT_TO_DINT(ot_stretch_need) THEN
                                ot_stretch_deficit := LINT_TO_DINT(ot_stretch_need);
                                ot_stretch_pending := TRUE;
                                ot_stretch_ok      := TRUE;
                              END_IF;
                            END_IF;
                          END_IF;
                        END_IF;
                      END_IF;
                    END_FOR;
                  END_IF;

                  IF ot_stretch_ok THEN
                    ot_idle_ok := TRUE;
                  ELSE
                    vOverlapConflict := TRUE;
                  END_IF;
                END_IF;
              END_IF;
            END_FOR;

  IF vOverlapConflict THEN vDestStn := 0; END_IF;
          END_IF;

          IF vDestStn > 0 THEN
            (* ── Commit idle-stretch: extend blocking batch CalTime ── *)
            IF vStretchPending THEN
              g_batch[vStretchUnitId].CalTime :=
                g_batch[vStretchUnitId].CalTime + vStretchDeficit;
              vStretchPending := FALSE;
            END_IF;

            (* ── Commit other-transporter idle-stretch ── *)
            IF ot_stretch_pending THEN
              g_batch[ot_stretch_unit_id].CalTime :=
                g_batch[ot_stretch_unit_id].CalTime + ot_stretch_deficit;
              ot_stretch_pending := FALSE;
            END_IF;

            IF ioTask[cov_t].Count < MAX_TASK_QUEUE THEN
              FOR sh := ioTask[cov_t].Count TO 1 BY -1 DO
                ioTask[cov_t].Queue[sh + 1] := ioTask[cov_t].Queue[sh];
              END_FOR;
              ioTask[cov_t].Queue[1].Unit         := ui;
              ioTask[cov_t].Queue[1].Stage        := 0;
              ioTask[cov_t].Queue[1].LiftStationTarget := vLoc;
              ioTask[cov_t].Queue[1].SinkStationTarget := vDestStn;
              ioTask[cov_t].Queue[1].StartTime   := vTaskStart;
              ioTask[cov_t].Queue[1].FinishTime  := vTaskEnd;
              ioTask[cov_t].Queue[1].CalcTime    := 0;
              ioTask[cov_t].Queue[1].MinTime     := 0;
              ioTask[cov_t].Queue[1].MaxTime     := 0;
              ioTask[cov_t].Queue[1].NttPrimary := 0;
              FOR si := 1 TO vDest.StationCount DO
                IF vDest.Stations[si] = vDestStn THEN
                  ioTask[cov_t].Queue[1].NttPrimary := 1;
                END_IF;
              END_FOR;
              ioTask[cov_t].Count := ioTask[cov_t].Count + 1;
              oDone := TRUE;
            END_IF;
          END_IF;

        END_IF; (* NOT vOnPrimary *)
      END_IF; (* vCovers + idle *)
      END_IF; (* NOT oDone *)
    END_FOR; (* transporter loop *)
    END_IF; (* NOT vAlready *)
  END_IF; (* valid target *)
END_FOR;

END_FUNCTION
